// TIA Portal V18 export
DATA_BLOCK "transfer_DB"   // DB1
VERSION : 0.1
// stored: AutoNumber true, DBAccessibleFromOPCUA true, InstanceOfName transfer, InstanceOfType FB
"transfer"
   // VAR
   //    ton_no_con { S7_SetPoint := 'True'} : TON_TIME;
   // END_VAR
BEGIN
END_DATA_BLOCK
